FUNCTION_BLOCK Recipe_10015_eineCookiebitte
VAR_INPUT
	execute	: BOOL;
	Order	: DUT_RECIPEORDER;
END_VAR
VAR_OUTPUT
	RecipeInfo	: DUT_RECIPEOFFER;
	RecipeDone	: BOOL;	
	InitDone	: BOOL;
END_VAR
VAR
	StepDone	: BOOL;
END_VAR

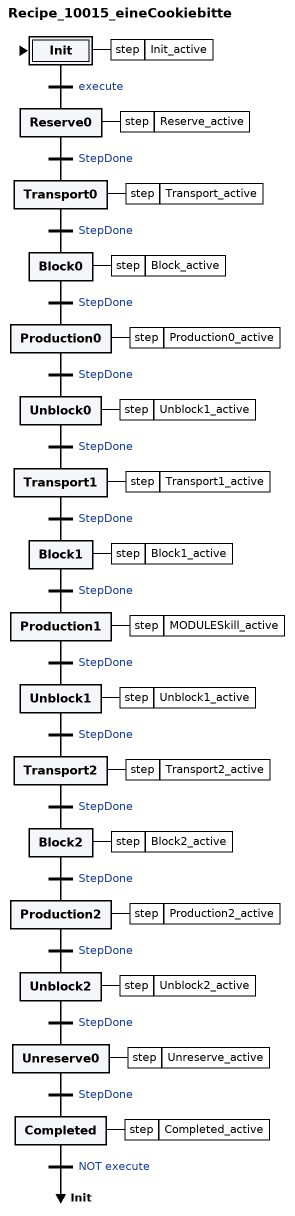
INITIAL_STEP Init:
    Init_active(N);  // step action
END_STEP
TRANSITION FROM Init TO Reserve0
    := execute;
END_TRANSITION
STEP Reserve0:
    Reserve_active(N);  // step action
END_STEP
TRANSITION FROM Reserve0 TO Transport0
    := StepDone;
END_TRANSITION
STEP Transport0:
    Transport_active(N);  // step action
END_STEP
TRANSITION FROM Transport0 TO Block0
    := StepDone;
END_TRANSITION
STEP Block0:
    Block_active(N);  // step action
END_STEP
TRANSITION FROM Block0 TO Production0
    := StepDone;
END_TRANSITION
STEP Production0:
    Production0_active(N);  // step action
END_STEP
TRANSITION FROM Production0 TO Unblock0
    := StepDone;
END_TRANSITION
STEP Unblock0:
    Unblock1_active(N);  // step action
END_STEP
TRANSITION FROM Unblock0 TO Transport1
    := StepDone;
END_TRANSITION
STEP Transport1:
    Transport1_active(N);  // step action
END_STEP
TRANSITION FROM Transport1 TO Block1
    := StepDone;
END_TRANSITION
STEP Block1:
    Block1_active(N);  // step action
END_STEP
TRANSITION FROM Block1 TO Production1
    := StepDone;
END_TRANSITION
STEP Production1:
    MODULESkill_active(N);  // step action
END_STEP
TRANSITION FROM Production1 TO Unblock1
    := StepDone;
END_TRANSITION
STEP Unblock1:
    Unblock1_active(N);  // step action
END_STEP
TRANSITION FROM Unblock1 TO Transport2
    := StepDone;
END_TRANSITION
STEP Transport2:
    Transport2_active(N);  // step action
END_STEP
TRANSITION FROM Transport2 TO Block2
    := StepDone;
END_TRANSITION
STEP Block2:
    Block2_active(N);  // step action
END_STEP
TRANSITION FROM Block2 TO Production2
    := StepDone;
END_TRANSITION
STEP Production2:
    Production2_active(N);  // step action
END_STEP
TRANSITION FROM Production2 TO Unblock2
    := StepDone;
END_TRANSITION
STEP Unblock2:
    Unblock2_active(N);  // step action
END_STEP
TRANSITION FROM Unblock2 TO Unreserve0
    := StepDone;
END_TRANSITION
STEP Unreserve0:
    Unreserve_active(N);  // step action
END_STEP
TRANSITION FROM Unreserve0 TO Completed
    := StepDone;
END_TRANSITION
STEP Completed:
    Completed_active(N);  // step action
END_STEP
TRANSITION FROM Completed TO Init
    := NOT execute;
END_TRANSITION

ACTION Block2_active:
StepDone := FALSE;

//Skill auswählen
ExecuteSkill.SkillID 		:= 1315;
ExecuteSkill.SkillName	 	:= 'Block';

//Parameter setzen

ExecuteSkill.Parameter[1].ID := 1;
ExecuteSkill.Parameter[1].Name := 'TaskID';
ExecuteSkill.Parameter[1].Value := 130;


(*
ExecuteSkill.Parameter[2].ID := ;
ExecuteSkill.Parameter[2].Name := '';
ExecuteSkill.Parameter[2].Value := ;
*)

(*
ExecuteSkill.Parameter[3].ID := ;
ExecuteSkill.Parameter[3].Name := '';
ExecuteSkill.Parameter[3].Value := ;
*)

(*
ExecuteSkill.Parameter[4].ID := ;
ExecuteSkill.Parameter[4].Name := '';
ExecuteSkill.Parameter[4].Value := ;
*)

(*
ExecuteSkill.Parameter[5].ID := ;
ExecuteSkill.Parameter[5].Name := '';
ExecuteSkill.Parameter[5].Value := ;
*)



ExecuteSkill();

StepDone := ExecuteSkill.Done;
END_ACTION

ACTION Unreserve_active:
StepDone := FALSE;

//Skill auswählen
ExecuteSkill.SkillID 		:= 1311;
ExecuteSkill.SkillName	 	:= 'Unreserve';

//Parameter setzen

ExecuteSkill.Parameter[1].ID := 1;
ExecuteSkill.Parameter[1].Name := 'TaskID';
ExecuteSkill.Parameter[1].Value := 131;


(*
ExecuteSkill.Parameter[2].ID := ;
ExecuteSkill.Parameter[2].Name := '';
ExecuteSkill.Parameter[2].Value := ;
*)

(*
ExecuteSkill.Parameter[3].ID := ;
ExecuteSkill.Parameter[3].Name := '';
ExecuteSkill.Parameter[3].Value := ;
*)

(*
ExecuteSkill.Parameter[4].ID := ;
ExecuteSkill.Parameter[4].Name := '';
ExecuteSkill.Parameter[4].Value := ;
*)

(*
ExecuteSkill.Parameter[5].ID := ;
ExecuteSkill.Parameter[5].Name := '';
ExecuteSkill.Parameter[5].Value := ;
*)



ExecuteSkill();

StepDone := ExecuteSkill.Done;
END_ACTION

ACTION Transport1_active:
StepDone := FALSE;

//Skill auswählen
ExecuteSkill.SkillID 		:= 1320;
ExecuteSkill.SkillName	 	:= 'Name';

//Parameter setzen

ExecuteSkill.Parameter[3].ID := 3;
ExecuteSkill.Parameter[3].Name := 'Velocity';
ExecuteSkill.Parameter[3].Value := 2500;



ExecuteSkill.Parameter[4].ID := 4 ;
ExecuteSkill.Parameter[4].Name := 'Acceleration';
ExecuteSkill.Parameter[4].Value := 1000 ;



ExecuteSkill.Parameter[1].ID := 1;
ExecuteSkill.Parameter[1].Name := 'TargetPosition X';
ExecuteSkill.Parameter[1].Value := 3200 ;
ExecuteSkill.Parameter[1].StringValue := '#DP#2#XPosition' ;




ExecuteSkill.Parameter[2].ID := 2;
ExecuteSkill.Parameter[2].Name := 'TargetPosition Z';
ExecuteSkill.Parameter[2].Value := 105;


(*
ExecuteSkill.Parameter[5].ID := ;
ExecuteSkill.Parameter[5].Name := '';
ExecuteSkill.Parameter[5].Value := ;
*)



ExecuteSkill();

StepDone := ExecuteSkill.Done;
END_ACTION

ACTION Block_active:
StepDone := FALSE;

//Skill auswählen
ExecuteSkill.SkillID 		:= 1315;
ExecuteSkill.SkillName	 	:= 'Block';

//Parameter setzen

ExecuteSkill.Parameter[1].ID := 1;
ExecuteSkill.Parameter[1].Name := 'TaskID';
ExecuteSkill.Parameter[1].Value := 124;


(*
ExecuteSkill.Parameter[2].ID := ;
ExecuteSkill.Parameter[2].Name := '';
ExecuteSkill.Parameter[2].Value := ;
*)

(*
ExecuteSkill.Parameter[3].ID := ;
ExecuteSkill.Parameter[3].Name := '';
ExecuteSkill.Parameter[3].Value := ;
*)

(*
ExecuteSkill.Parameter[4].ID := ;
ExecuteSkill.Parameter[4].Name := '';
ExecuteSkill.Parameter[4].Value := ;
*)

(*
ExecuteSkill.Parameter[5].ID := ;
ExecuteSkill.Parameter[5].Name := '';
ExecuteSkill.Parameter[5].Value := ;
*)



ExecuteSkill();

StepDone := ExecuteSkill.Done;
END_ACTION

ACTION Block1_active:
StepDone := FALSE;

//Skill auswählen
ExecuteSkill.SkillID 		:= 1315;
ExecuteSkill.SkillName	 	:= 'Block';

//Parameter setzen

ExecuteSkill.Parameter[1].ID := 1;
ExecuteSkill.Parameter[1].Name := 'TaskID';
ExecuteSkill.Parameter[1].Value := 127;


(*
ExecuteSkill.Parameter[2].ID := ;
ExecuteSkill.Parameter[2].Name := '';
ExecuteSkill.Parameter[2].Value := ;
*)

(*
ExecuteSkill.Parameter[3].ID := ;
ExecuteSkill.Parameter[3].Name := '';
ExecuteSkill.Parameter[3].Value := ;
*)

(*
ExecuteSkill.Parameter[4].ID := ;
ExecuteSkill.Parameter[4].Name := '';
ExecuteSkill.Parameter[4].Value := ;
*)

(*
ExecuteSkill.Parameter[5].ID := ;
ExecuteSkill.Parameter[5].Name := '';
ExecuteSkill.Parameter[5].Value := ;
*)



ExecuteSkill();

StepDone := ExecuteSkill.Done;
END_ACTION

ACTION Unblock2_active:
StepDone := FALSE;

//Skill auswählen
ExecuteSkill.SkillID 		:= 1316;
ExecuteSkill.SkillName	 	:= 'Unblock';

//Parameter setzen

ExecuteSkill.Parameter[1].ID := 1;
ExecuteSkill.Parameter[1].Name := 'TaskID';
ExecuteSkill.Parameter[1].Value := 131;


(*
ExecuteSkill.Parameter[2].ID := ;
ExecuteSkill.Parameter[2].Name := '';
ExecuteSkill.Parameter[2].Value := ;
*)

(*
ExecuteSkill.Parameter[3].ID := ;
ExecuteSkill.Parameter[3].Name := '';
ExecuteSkill.Parameter[3].Value := ;
*)

(*
ExecuteSkill.Parameter[4].ID := ;
ExecuteSkill.Parameter[4].Name := '';
ExecuteSkill.Parameter[4].Value := ;
*)

(*
ExecuteSkill.Parameter[5].ID := ;
ExecuteSkill.Parameter[5].Name := '';
ExecuteSkill.Parameter[5].Value := ;
*)



ExecuteSkill();

StepDone := ExecuteSkill.Done;
END_ACTION

ACTION Completed_active:
RecipeDone := TRUE;
StepDone := FALSE;
END_ACTION

ACTION Unblock_active:
StepDone := FALSE;

//Skill auswählen
ExecuteSkill.SkillID 		:= 1316;
ExecuteSkill.SkillName	 	:= 'Unblock';

//Parameter setzen

ExecuteSkill.Parameter[1].ID := 1;
ExecuteSkill.Parameter[1].Name := 'TaskID';
ExecuteSkill.Parameter[1].Value := 125;


(*
ExecuteSkill.Parameter[2].ID := ;
ExecuteSkill.Parameter[2].Name := '';
ExecuteSkill.Parameter[2].Value := ;
*)

(*
ExecuteSkill.Parameter[3].ID := ;
ExecuteSkill.Parameter[3].Name := '';
ExecuteSkill.Parameter[3].Value := ;
*)

(*
ExecuteSkill.Parameter[4].ID := ;
ExecuteSkill.Parameter[4].Name := '';
ExecuteSkill.Parameter[4].Value := ;
*)

(*
ExecuteSkill.Parameter[5].ID := ;
ExecuteSkill.Parameter[5].Name := '';
ExecuteSkill.Parameter[5].Value := ;
*)



ExecuteSkill();

StepDone := ExecuteSkill.Done;
END_ACTION

ACTION Production2_active:
StepDone := FALSE;
RecipeDone := FALSE;
//Skill auswählen
ExecuteSkill.SkillID 		:= 1339;
ExecuteSkill.SkillName	 	:= 'ParameterTESTSKILL1339';


ExecuteSkill.Parameter[0].ID := 10;
ExecuteSkill.Parameter[0].Name := 'Blinkfrequenz';
ExecuteSkill.Parameter[0].Value := Order.UserParameter[0].Value*2;


ExecuteSkill();

StepDone := ExecuteSkill.Done;
END_ACTION

ACTION Init_active:
RecipeDone := FALSE;

// Initialisation of Recipe Parameters an name etc
RecipeInfo.Name := 'one cookie please';
RecipeInfo.Description := 'Order one cookie and do testskills before and after';
RecipeInfo.Dummy := FALSE;
RecipeInfo.RecipeID := 10015; 	// 
Initdone := TRUE;

//Parameter 0:

	RecipeInfo.UserParameter[0].Dummy 		:= FALSE;
	RecipeInfo.UserParameter[0].Default		:= 0.5;
	RecipeInfo.UserParameter[0].Description	:= 'Recipe BLinkgeschwindigkeit';
	RecipeInfo.UserParameter[0].MaxValue	:= 50.0;
	RecipeInfo.UserParameter[0].MinValue	:= 0;
	RecipeInfo.UserParameter[0].Name		:= 'Production Frequenz';
	RecipeInfo.UserParameter[0].Unit		:= 'HZ';

//Parameter 1:
(*
	RecipeInfo.UserParameter[1].Dummy 		:= 
	RecipeInfo.UserParameter[1].Default		:=
	RecipeInfo.UserParameter[1].Description	:=
	RecipeInfo.UserParameter[1].MaxValue	:=
	RecipeInfo.UserParameter[1].MinValue	:=
	RecipeInfo.UserParameter[1].Name		:=
	RecipeInfo.UserParameter[1].Unit		:=
*)
	

//Parameter 2:

(*
	RecipeInfo.UserParameter[2].Dummy 		:= 
	RecipeInfo.UserParameter[2].Default		:=
	RecipeInfo.UserParameter[2].Description	:=
	RecipeInfo.UserParameter[2].MaxValue	:=
	RecipeInfo.UserParameter[2].MinValue	:=
	RecipeInfo.UserParameter[2].Name		:=
	RecipeInfo.UserParameter[2].Unit		:=
*)

//Parameter 3:

(*
	RecipeInfo.UserParameter[3].Dummy 		:= 
	RecipeInfo.UserParameter[3].Default		:=
	RecipeInfo.UserParameter[3].Description	:=
	RecipeInfo.UserParameter[3].MaxValue	:=
	RecipeInfo.UserParameter[3].MinValue	:=
	RecipeInfo.UserParameter[3].Name		:=
	RecipeInfo.UserParameter[3].Unit		:=
*)

//Parameter 4:

(*
	RecipeInfo.UserParameter[4].Dummy 		:= 
	RecipeInfo.UserParameter[4].Default		:=
	RecipeInfo.UserParameter[4].Description	:=
	RecipeInfo.UserParameter[4].MaxValue	:=
	RecipeInfo.UserParameter[4].MinValue	:=
	RecipeInfo.UserParameter[4].Name		:=
	RecipeInfo.UserParameter[4].Unit		:=
*)


//Parameter 5:

(*
	RecipeInfo.UserParameter[5].Dummy 		:= 
	RecipeInfo.UserParameter[5].Default		:=
	RecipeInfo.UserParameter[5].Description	:=
	RecipeInfo.UserParameter[5].MaxValue	:=
	RecipeInfo.UserParameter[5].MinValue	:=
	RecipeInfo.UserParameter[5].Name		:=
	RecipeInfo.UserParameter[5].Unit		:=
*)
END_ACTION

ACTION Transport2_active:
StepDone := FALSE;

//Skill auswählen
ExecuteSkill.SkillID 		:= 1320;
ExecuteSkill.SkillName	 	:= 'Transport';

//Parameter setzen

ExecuteSkill.Parameter[3].ID := 3;
ExecuteSkill.Parameter[3].Name := 'Velocity';
ExecuteSkill.Parameter[3].Value := 2800;



ExecuteSkill.Parameter[1].ID :=  1;
ExecuteSkill.Parameter[1].Name := 'TargetPosition X';
ExecuteSkill.Parameter[1].Value := 30 ;
ExecuteSkill.Parameter[1].StringValue := '#DP#2#XPosition';



ExecuteSkill.Parameter[2].ID := 2;
ExecuteSkill.Parameter[2].Name := 'TargetPosition Z';
ExecuteSkill.Parameter[2].Value := 0 ;



ExecuteSkill.Parameter[4].ID := 4;
ExecuteSkill.Parameter[4].Name := 'Acceleration';
ExecuteSkill.Parameter[4].Value := 2000 ;


(*
ExecuteSkill.Parameter[5].ID := ;
ExecuteSkill.Parameter[5].Name := '';
ExecuteSkill.Parameter[5].Value := ;
*)



ExecuteSkill();

StepDone := ExecuteSkill.Done;
END_ACTION

ACTION MODULESkill_active:
StepDone := FALSE;
RecipeDone := FALSE;
//Skill auswählen
ExecuteSkill.SkillID 		:= 1010;
ExecuteSkill.SkillName	 	:= 'Cookie ausgeben';





ExecuteSkill();

StepDone := ExecuteSkill.Done;
END_ACTION

ACTION Reserve_active:
StepDone := FALSE;
RecipeDone := FALSE;
//Skill auswählen
ExecuteSkill.SkillID 		:= 1310;
ExecuteSkill.SkillName	 	:= 'Reserve';

//Parameter setzen

ExecuteSkill.Parameter[1].ID := 1;
ExecuteSkill.Parameter[1].Name := 'TaskID';
ExecuteSkill.Parameter[1].Value := 123;


(*
ExecuteSkill.Parameter[2].ID := ;
ExecuteSkill.Parameter[2].Name := '';
ExecuteSkill.Parameter[2].Value := ;
*)

(*
ExecuteSkill.Parameter[3].ID := ;
ExecuteSkill.Parameter[3].Name := '';
ExecuteSkill.Parameter[3].Value := ;
*)

(*
ExecuteSkill.Parameter[4].ID := ;
ExecuteSkill.Parameter[4].Name := '';
ExecuteSkill.Parameter[4].Value := ;
*)

(*
ExecuteSkill.Parameter[5].ID := ;
ExecuteSkill.Parameter[5].Name := '';
ExecuteSkill.Parameter[5].Value := ;
*)



ExecuteSkill();

StepDone := ExecuteSkill.Done;
END_ACTION

ACTION Production0_active:
StepDone := FALSE;
RecipeDone := FALSE;
//Skill auswählen
ExecuteSkill.SkillID 		:= 1337;
ExecuteSkill.SkillName	 	:= 'Testmodul1';

ExecuteSkill();

StepDone := ExecuteSkill.Done;
END_ACTION

ACTION Unblock1_active:
StepDone := FALSE;

//Skill auswählen
ExecuteSkill.SkillID 		:= 1316;
ExecuteSkill.SkillName	 	:= 'Unblock';

//Parameter setzen

ExecuteSkill.Parameter[1].ID := 1;
ExecuteSkill.Parameter[1].Name := 'TaskID';
ExecuteSkill.Parameter[1].Value := 128 ;


(*
ExecuteSkill.Parameter[2].ID := ;
ExecuteSkill.Parameter[2].Name := '';
ExecuteSkill.Parameter[2].Value := ;
*)

(*
ExecuteSkill.Parameter[3].ID := ;
ExecuteSkill.Parameter[3].Name := '';
ExecuteSkill.Parameter[3].Value := ;
*)

(*
ExecuteSkill.Parameter[4].ID := ;
ExecuteSkill.Parameter[4].Name := '';
ExecuteSkill.Parameter[4].Value := ;
*)

(*
ExecuteSkill.Parameter[5].ID := ;
ExecuteSkill.Parameter[5].Name := '';
ExecuteSkill.Parameter[5].Value := ;
*)



ExecuteSkill();

StepDone := ExecuteSkill.Done;
END_ACTION

ACTION Transport_active:
StepDone := FALSE;

//Skill auswählen
ExecuteSkill.SkillID 		:= 1320;
ExecuteSkill.SkillName	 	:= 'Transport';

//Parameter setzen

ExecuteSkill.Parameter[3].ID :=3 ;
ExecuteSkill.Parameter[3].Name := 'Velocity';
ExecuteSkill.Parameter[3].Value := 1500;



ExecuteSkill.Parameter[1].ID :=1 ;
ExecuteSkill.Parameter[1].Name := 'TargetPosition X';
ExecuteSkill.Parameter[1].StringValue := '#DP#2#XPosition';
ExecuteSkill.Parameter[1].Value := 200 ;


ExecuteSkill.Parameter[2].ID := 2 ;
ExecuteSkill.Parameter[2].Name := 'TargetPosition Z';
ExecuteSkill.Parameter[2].Value := 70 ;



ExecuteSkill.Parameter[4].ID := 4 ;
ExecuteSkill.Parameter[4].Name := 'Acceleration';
ExecuteSkill.Parameter[4].Value := 4500;


(*
ExecuteSkill.Parameter[5].ID := ;
ExecuteSkill.Parameter[5].Name := '';
ExecuteSkill.Parameter[5].Value := ;
*)



ExecuteSkill();

StepDone := ExecuteSkill.Done;
END_ACTION

END_FUNCTION_BLOCK

(* stored: Version 1.1.0.1, ProductVersion 3.1.0.25
   POU Recipe_10015_eineCookiebitte: Id {d20aaa89-4044-4a5b-8325-f92b7bb75a3d}
   Action Block2_active: Id {010742ed-ef32-43ef-a2d4-c353f9f23a3d}
   Action Unreserve_active: Id {4fe15935-0862-434c-8658-57b75d607287}
   Action Transport1_active: Id {51a389a3-0412-486f-a691-d18a94026076}
   Action Block_active: Id {60d655ca-6f30-4965-b69a-f83038665152}
   Action Block1_active: Id {65de957a-1764-4adc-b3a2-d6af946a6e82}
   Action Unblock2_active: Id {7576cafb-2267-47dd-92e2-207be403dcd6}
   Action Completed_active: Id {76e5acc0-7a0b-454f-a5aa-0af697c3dca1}
   Action Unblock_active: Id {7dedbf59-e321-489f-9e3e-753539c802e0}
   Action Production2_active: Id {7ed35672-f953-4b63-b113-0dc500636b99}
   Action Init_active: Id {80ae27d1-f725-4e81-89a3-b7b8d50bb5c5}
   Action Transport2_active: Id {86cbf88e-00bf-4007-b6e8-b37e3235b60d}
   Action MODULESkill_active: Id {962c7458-b578-48bb-86bb-04e43b0bd1d1}
   Action Reserve_active: Id {a6a523a9-0ce4-4ef1-aaa5-409d10c6f825}
   Action Production0_active: Id {aa3b3b50-390d-4c1f-b463-14e6b37ad61b}
   Action Unblock1_active: Id {ab8c0b41-1dc6-479a-ad6c-0b0cea8e2aaf}
   Action Transport_active: Id {c411c5b3-7657-4eeb-b107-fcdf8977ae57} *)
